Staubli VAL3: socketServer.dtx

mdesc nom_speed = {rmax=9999, blend=off}
sio sioSocket = {link=Socket\HelloServer}
num nNum
num nBuffer
string sBuffer
string sInput[50]
num nFailCounter
jointRx jTest
pointRs pPointRs = {fatherId=world[0]}
bool bDetectInput
tool tClaw = {z=90, fatherId=flange[0], ioLink=valve1}
bool bClawClosed
num nMovementData[3]
